// TwinCAT 3 PLC project PLC
// ProgramVersion: 3.1.4026.19
// libraries:
//   SPT Base Types, * (Beckhoff Automation LLC)
//   SPT Components, * (Beckhoff Automation LLC)
//   SPT Diagnostic, * (Beckhoff Automation LLC)
//   SPT EtherCat, * (Beckhoff Automation LLC)
//   SPT Event Logger, * (Beckhoff Automation LLC)
//   SPT Motion Control, * (Beckhoff Automation LLC)
//   SPT Utilities, * (Beckhoff Automation LLC)
//   Tc2_MC2, * (Beckhoff Automation GmbH)
//   Tc2_Standard, * (Beckhoff Automation GmbH)
//   Tc2_System, * (Beckhoff Automation GmbH)
//   Tc3_EventLogger, * (Beckhoff Automation GmbH)
//   Tc3_Module, * (Beckhoff Automation GmbH)
//   Tc3_PackML_V3, * (Beckhoff Automation GmbH)
// project tree:
//   / GlobalTextList.TcGTLO, PlcTask.TcTTO, Visualization Manager.TcVMO (not stored)
//   POUs/Function Blocks/Reversing Sequence/ E_RevSeq.TcDUT, ReversingSequence.TcPOU
//   POUs/ MAIN.TcPOU
//   POUs/Modules/00 Machine/ Machine.TcPOU
//   VISUs/ Visualization.TcVIS
// real-time tasks:
//   TASK PlcTask: cycle T#10ms, priority 20, ADS port 350
// motion (NC):
//   TASK NC-Task 1 SAF: cycle T#2ms, priority 4, ADS port 501
//   TASK NC-Task 1 SVB: cycle T#10ms, priority 8, ADS port 511
//   AXIS Axis 1 (id 1)
//     OtherSettings: AllowMotionCmdToSlave=true
//     encoder EncType=1
//       EncPara: ScaleFactorNumerator=1
//         SoftEndMaxControl: Enable=true, Range=100
//     drive DrvType=5
//       Analog: TorqueSetpointScale=10, ScaleFactorActTorque=0.1
//     controller CtrType=1
//       CtrPara: PriorControlFactor=1
//         Observer: BandWidth=20
// variable links:
//   PLC/PLC Instance <-> NC-Task 1 SAF/Axes/Axis 1
//     PlcTask Inputs/MAIN.Machine.VAxis.BasicAxis._Axis.NcToPlc <-> Outputs/ToPlc
//     PlcTask Outputs/MAIN.Machine.VAxis.BasicAxis._Axis.PlcToNc <-> Inputs/FromPlc

CONFIGURATION PLC
    RESOURCE PLC ON TwinCAT3
        TASK PlcTask(INTERVAL := T#10ms, PRIORITY := 20);
        PROGRAM MAIN WITH PlcTask : MAIN;
    END_RESOURCE
END_CONFIGURATION

// ---- POUs/Function Blocks/Reversing Sequence/E_RevSeq.TcDUT
TYPE E_RevSeq : (
		Stopped,
		Move1,
		Wait1,
		Idle1,
		Move2,
		Wait2,
		Idle2,
		Error
	) INT;
END_TYPE

// ---- POUs/MAIN.TcPOU
PROGRAM MAIN
VAR
	Machine : Machine := (Name := 'Machine');
END_VAR

(*All sample code provided by Beckhoff Automation LLC are for illustrative purposes only and are provided “as is” and without any warranties, express or implied. Actual implementations in applications will vary significantly. Beckhoff Automation LLC shall have no liability for, and does not waive any rights in relation to, any code samples that it provides or the use of such code samples for any purpose.*)

(*
	The FB_Component_BasicAxis has all of the basic moves provided by the MC2 library built in;
	however, by use of the strategy pattern more complex move sequences can be programmed externally and an instance of those function blocks can be passed into the FB_Component_BasicAxis.ExternalSequence property.
	Setting the property 'ExternalSequence' to the instance of a function block that implements the I_MotionSequence interface will allow for the RunExternalSequence method to execute that code.
	While it is typical to set the HomeMethod or ResetMethod in an initialization routine and then not change it, the ExternalSequence can be changed as often as needed.

	Note: After setting the ExternalSequence property, a call to the Axis's CyclicLogic method is required before it can be used. This can be done by either allowing 1 PLC scan between setting the ExternalSequence property
	and the call to the RunExternalSequence method, or by calling the CyclicLogic method directly after setting the ExternalSequence.

	When creating your own external sequence, it is best to start by using a state machine within the CyclicLogic method and use the Execute method to move the state machine from idle to the first step.
		
	Stopping the external sequence requires some consideration related to its internal state machine. The example for a Reversing Sequence given in this project never has an end point and will continue its sequence indefinitely.
	Because the FB_Component_BasicAxis.Stop method calls an instance of MC_Halt internally, the axis might stop momentarily but will ultimately start again once the timers have elasped.
	To stop the reversing sequence an additional Stop method was added that calls the Axis.Stop method and sets the state machine to idle, in order to prevent it from restarting.

 


*)

//This is for debug only and should be removed
_AppInfo.KeepOutputsOnBP := TRUE;

//
Machine.CyclicLogic();

END_PROGRAM

// ---- POUs/Modules/00 Machine/Machine.TcPOU
FUNCTION_BLOCK Machine EXTENDS FB_PackML_BaseModule
VAR
	VAxis		  : FB_Component_BasicAxis := (Name := 'V Axis');
	RevSequence	  : ReversingSequence;
	startRevSeq	  : BOOL;
	stopAxis	  : BOOL;
	moveAbs		  : BOOL;
	abortExternal : BOOL;
END_VAR

METHOD PUBLIC CyclicLogic
VAR
END_VAR
IF NOT _InitComplete THEN
	_InitComplete := Initialize();
	RETURN;
END_IF

SUPER^.CyclicLogic();
END_METHOD

METHOD PROTECTED Execute
VAR
END_VAR
RevSequence.Velocity  := 5.0;
RevSequence.Position1 := 10.0;
RevSequence.IdleTime  := 1000;
RevSequence.Position2 := 0.0;

//Test Reversing Sequence
IF startRevSeq THEN
	startRevSeq			   := FALSE;
	VAXis.ExternalSequence := RevSequence;
	VAxis.CyclicLogic(); //Update the internals before calling the method
	VAxis.RunExternalSequence();
END_IF

//Properly stops the External Sequence
IF stopAxis THEN
	stopAxis := FALSE;
	RevSequence.Stop();
END_IF

//Aborts the existing move, starts new move, but ultimately returns to the External Sequence
IF moveAbs THEN
	moveAbs := FALSE;
	VAxis.MoveAbsolute(Position := 100.0, AbortPrevious := TRUE);
END_IF

//Halts the axis, but not the state machine of the External Sequence
IF abortExternal THEN
	abortExternal := FALSE;
	IF VAxis.Stop() THEN
		;
	END_IF
END_IF
END_METHOD

// Automatically enables and disables HMI control based on the PackML mode
METHOD PROTECTED HMIPermissions

// This method is called cyclically by CyclicLogic()
AllowHMIControl(ThisModuleOnly := TRUE);
END_METHOD

METHOD PROTECTED Initialize : BOOL;
VAR
END_VAR
Initialize := FALSE;
CASE DescendantSequenceState OF
	0:
		RegisterComponent(Component := VAxis);
		DescendantSequenceState := DescendantSequenceState + 10;

	10:
		IF SUPER^.Initialize() THEN
			Initialize := TRUE;
		END_IF
END_CASE
END_METHOD

METHOD PROTECTED Starting
VAR
END_VAR
CASE SequenceState OF
	0:
		NoStateTasksToComplete := FALSE;
		SequenceState		   := SequenceState + 10;

	10:
		IF VAxis.Enable() THEN
			SequenceState := SequenceState + 10;
		END_IF

	20:
		IF VAxis.Enabled THEN
			SequenceState := SequenceState + 10;
		END_IF

	30:
		StateTasksComplete := TRUE;
END_CASE

SUPER^.Starting();
END_METHOD

END_FUNCTION_BLOCK

// ---- POUs/Function Blocks/Reversing Sequence/ReversingSequence.TcPOU
FUNCTION_BLOCK ReversingSequence EXTENDS FB_CyclicFB IMPLEMENTS I_MotionSequence
VAR
	_Axis		 : I_BasicAxis;
	_Position1	 : LREAL;
	_Position2	 : LREAL;
	_Velocity	 : LREAL;
	_IdleTime	 : INT;
	fbMove		 : MC_MoveAbsolute;
	fbIdle		 : TON;
	SequenceStep : E_RevSeq;
END_VAR

{warning 'add property implementation'}
PROPERTY Axis : SPT_Motion_Control.I_BasicAxis
GET
Axis := _Axis;
END_GET
SET
_Axis := Axis;
END_SET
END_PROPERTY

{warning 'add method implementation '}
METHOD CyclicLogic
CASE SequenceStep OF
	E_RevSeq.Stopped: //Idle, waiting for Execute method
	E_RevSeq.Move1:	  //Move to Position 1
		fbMove(Axis		:= _Axis.Axis,
			   Execute	:= TRUE,
			   Position := _Position1,
			   Velocity := _Velocity);

		SequenceStep := E_RevSeq.Wait1;

	E_RevSeq.Wait1:
		fbMove(Axis := _Axis.Axis, Execute := FALSE);
		IF NOT fbmove.Busy THEN
			IF NOT fbMove.Error THEN
				SequenceStep := E_RevSeq.Idle1;
			ELSE
				_ErrorID	 := 11;
				SequenceStep := E_RevSeq.Error;
			END_IF
		END_IF

	E_RevSeq.Idle1: //Wait for idle time
		fbIdle(IN := TRUE, PT := TO_TIME(_IdleTime));
		IF fbIdle.Q THEN
			fbIdle(IN := FALSE);
			SequenceStep := E_RevSeq.Move2;
		END_IF

	E_RevSeq.Move2: //Move to Posotion 2
		fbMove(Axis		:= _Axis.Axis,
			   Execute	:= TRUE,
			   Position := _Position2,
			   Velocity := _Velocity);

		SequenceStep := E_RevSeq.Wait2;

	E_RevSeq.Wait2:
		fbMove(Axis := _Axis.Axis, Execute := FALSE);
		IF NOT fbmove.Busy THEN
			IF NOT fbMove.Error THEN
				SequenceStep := E_RevSeq.Idle2;
			ELSE
				_ErrorID	 := 11;
				SequenceStep := E_RevSeq.Error;
			END_IF
		END_IF

	E_RevSeq.Idle2: //Wait for Idle time
		fbIdle(IN := TRUE, PT := TO_TIME(_IdleTime));
		IF fbIdle.Q THEN
			fbIdle(IN := FALSE);
			SequenceStep := E_RevSeq.Move1;
		END_IF

	E_RevSeq.Error: //Error Step
		_Error := TRUE;
END_CASE

_Busy := SequenceStep <> 0;
END_METHOD

{warning 'add method implementation '}
METHOD Execute : BOOL
IF (_Axis = 0) OR _Busy THEN
	RETURN;
END_IF

_Busy		 := TRUE;
_Error		 := FALSE;
_ErrorID	 := 0;
SequenceStep := E_RevSeq.Move1;
Execute		 := TRUE;
END_METHOD

PROPERTY IdleTime : INT
GET
IdleTime := _IdleTime;
END_GET
SET
_IdleTime := IdleTime;
END_SET
END_PROPERTY

PROPERTY Position1 : LREAL
GET
Position1 := _Position1;
END_GET
SET
_Position1 := Position1;
END_SET
END_PROPERTY

PROPERTY Position2 : LREAL
GET
Position2 := _Position2;
END_GET
SET
_Position2 := Position2;
END_SET
END_PROPERTY

METHOD Stop : BOOL
VAR_INPUT
END_VAR
Stop := FALSE;
IF _Axis <> 0 THEN
	SequenceStep := E_RevSeq.Stopped;
	IF _Axis.Stop() THEN
		Stop := TRUE;
	END_IF
END_IF
END_METHOD

PROPERTY Velocity : LREAL
GET
Velocity := _Velocity;
END_GET
SET
_Velocity := Velocity;
END_SET
END_PROPERTY

END_FUNCTION_BLOCK

// ---- VISUs/Visualization.TcVIS
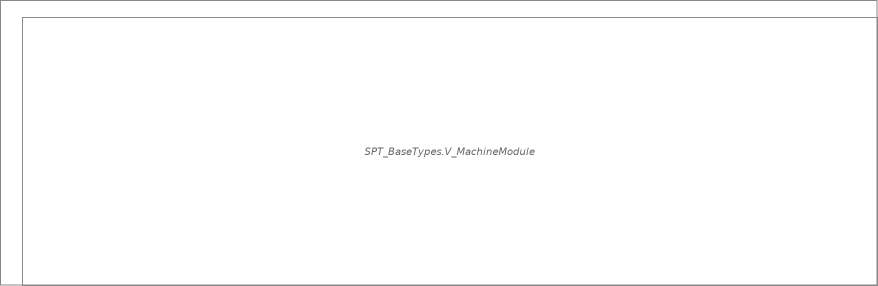
VISUALIZATION Visualization  // 878x286
    Frame (22,17 856x269)
        shows SPT_BaseTypes.V_MachineModule(HMI := MAIN.Machine.PackMLBaseModule_HMI)
END_VISUALIZATION
